FUNCTION_BLOCK FB_ScrollPump
VAR_IN_OUT
	iq_stPFO	:	ST_RoughPump;
END_VAR
VAR_INPUT
	TurboIsON : BOOL;
	VentValve	: ST_VCC_NO;
END_VAR
VAR
	Tmr_TOF : TOF;
	//Previous_RunSW : BOOL;
END_VAR

//Turn on scroll pump if the Turbo Vent Valve is closed. So you are not just
// pumping air and accomplishing nothing

// cannot turn off scroll pump if turb is running. delay scroll off 150s.  


Tmr_TOF(IN:=TurboIsON, PT := T#150S);

IF VentValve.xCLS_DO THEN
	iq_stPFO.q_xRunDo := (Tmr_TOF.Q OR iq_stPFO.i_xRunSW);
ELSE
	iq_stPFO.q_xRunDo := FALSE;
END_IF

iq_stPFO.i_xRunSW := iq_stPFO.q_xRunDo;

END_FUNCTION_BLOCK

(* stored: Version 1.1.0.1, ProductVersion 3.1.4020.12
   POU FB_ScrollPump: Id {95800034-a8e9-430e-af6e-1fa7a649fe90}, SpecialFunc None *)
